(* IEC 61131-3 sources: CodesysTest/export/UN00 - Sharp Bagger/EM02 - Discharge/EM02_Discharge.pou, 2 files *)

(* ---- EM02_Discharge.pou.st ---- *)
(*#-#-#-#-#-#-#-#-#-#---Declaration---#-#-#-#-#-#-#-#-#-#-#-#-#*)

FUNCTION_BLOCK EM02_Discharge EXTENDS FB_PackMLStates IMPLEMENTS IEM02_Discharge
VAR_INPUT
END_VAR
VAR_OUTPUT
END_VAR
VAR
END_VAR
(*#-#-#-#-#-#-#-#-#-#---Implementation---#-#-#-#-#-#-#-#-#-#-#-#-#*)

(* ---- TakeAwayBag.m.st ---- *)
(*#-#-#-#-#-#-#-#-#-#---Declaration---#-#-#-#-#-#-#-#-#-#-#-#-#*)

{warning 'add method implementation '}
METHOD TakeAwayBag
VAR_INPUT
		caller : IAllObjects;
END_VAR
(*#-#-#-#-#-#-#-#-#-#---Implementation---#-#-#-#-#-#-#-#-#-#-#-#-#*)
